// Mitsubishi GX Works2 project: 240930_공급가공분배2   PLC: Q03UDV

PROGRAM MAIN
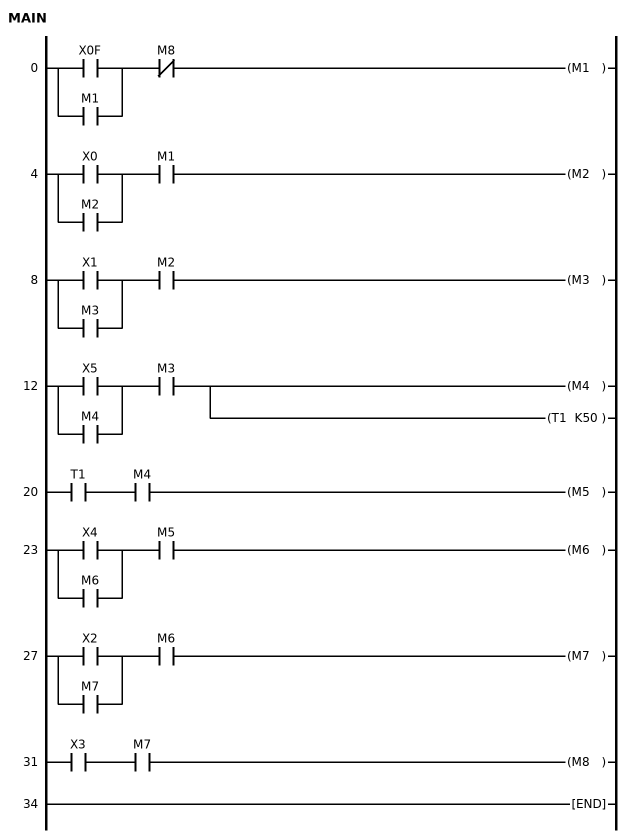
0     LD      X0F
      OR      M1
      ANI     M8
      OUT     M1
4     LD      X0
      OR      M2
      AND     M1
      OUT     M2
8     LD      X1
      OR      M3
      AND     M2
      OUT     M3
12    LD      X5
      OR      M4
      AND     M3
      OUT     M4
      OUT     T1 K50
20    LD      T1
      AND     M4
      OUT     M5
23    LD      X4
      OR      M6
      AND     M5
      OUT     M6
27    LD      X2
      OR      M7
      AND     M6
      OUT     M7
31    LD      X3
      AND     M7
      OUT     M8
34    END
END_PROGRAM

PROGRAM OUTPUT
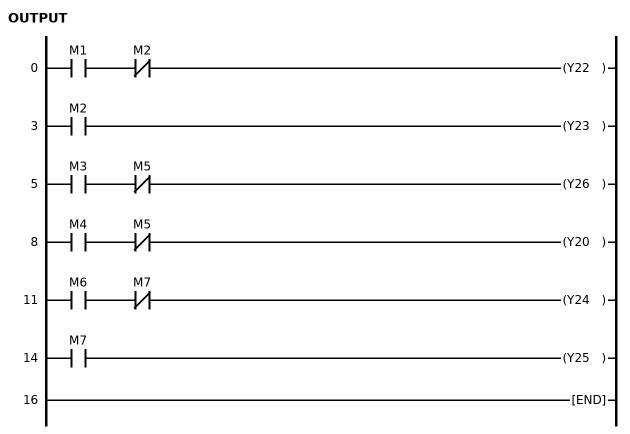
0     LD      M1
      ANI     M2
      OUT     Y22
3     LD      M2
      OUT     Y23
5     LD      M3
      ANI     M5
      OUT     Y26
8     LD      M4
      ANI     M5
      OUT     Y20
11    LD      M6
      ANI     M7
      OUT     Y24
14    LD      M7
      OUT     Y25
16    END
END_PROGRAM
